{attribute 'qualified_only'}
VAR_GLOBAL CONSTANT
    cHR_SuccesDone : HRESULT := 16#20000001; //Successfully done
    cHR_SuccesBusy : HRESULT := 16#20000002; //Busy, keep calling to wait for done or error    
END_VAR

(* stored: Version 1.1.0.1, ProductVersion 3.1.4019.2
   GVL GVL_HResultSuccess: Id {c39dda62-3ed3-43c5-989a-31eb429e44df} *)
